FUNCTION_BLOCK TcoDaqTestContext EXTENDS TcoCore._internals_TcoContext
VAR
	_sut : TcoDaqImplementationTest(THIS^);
	_msg : TcoDaqData;	
END_VAR

METHOD PROTECTED Main
VAR 
	_index : INT;
	_sb : TcoCore.StringBuilder;
END_VAR
CASE _testId OF     
    eTcoDaqTests.Push:
		_sut.Push(ADR(_msg));			 		
END_CASE

_sut();
END_METHOD

END_FUNCTION_BLOCK

(* stored: Version 1.1.0.1
   POU TcoDaqTestContext: Id {4b623250-6d62-0909-057c-b6bc6710b45c}, SpecialFunc None
   Method Main: Id {a93cd5b9-c57e-0b8b-0495-ebbc2998977f} *)
